(* PLC project PLC, Beckhoff Automation GmbH TwinCAT PLC Control 3.5.20.60 *)
(* stored: creationDateTime 2026-07-21T08:44:33.9440189, modificationDateTime 2026-07-21T08:44:33.9440189 *)

TYPE ST_ADS_API_ScadaViewerApp_PLC_Out_Status_Boxes :

STRUCT

	Presence				:	ARRAY [1..6] OF BOOL;	// |1| Přítomnsot boxu 1-6
	Full					:	ARRAY [1..6] OF BOOL;	// |2| Zaúlnění boxu 1-6
	Count					:	ARRAY [1..6] OF UINT;	// |3| Počet v boxu 1-6
	
END_STRUCT

END_TYPE
